// Mitsubishi GX Works2 project: PLS_programfiler_v1.0   PLC: FX2N/FX2NC

// global labels: Global1
VAR_GLOBAL
  Temperaturliste AT D0 : ARRAY [0..49] OF INT;
END_VAR

// task Task_01 (event TRUE, interval 0, priority 31): 

PROGRAM Kap7_765
(* structured ladder/FBD written out as ST: instructions are called as NAME(EN, inputs, outputs); _pN, _eN, _tN stand for wires *)
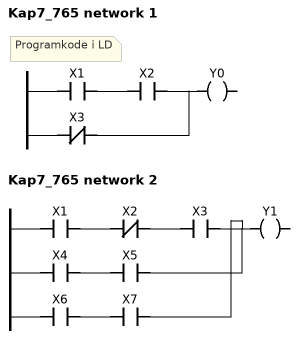
(* network 1 *)
(* Programkode i LD *)
Y0 := (X1 AND X2) OR (NOT X3);
(* network 2 *)
Y1 := (X1 AND NOT X2 AND X3) OR (X4 AND X5) OR (X6 AND X7);
END_PROGRAM

PROGRAM Kap7_766
(* structured ladder/FBD written out as ST: instructions are called as NAME(EN, inputs, outputs); _pN, _eN, _tN stand for wires *)
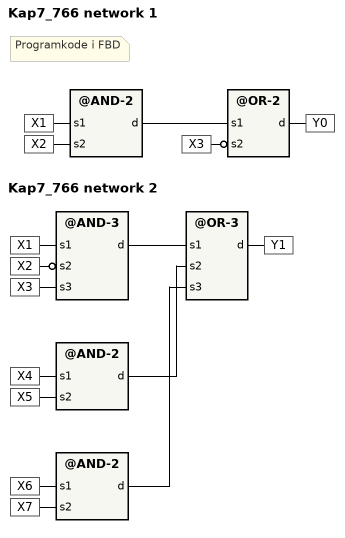
(* network 1 *)
(* Programkode i FBD *)
Y0 := @OR-2(@AND-2(X1, X2), NOT X3);
(* network 2 *)
Y1 := @OR-3(@AND-3(X1, NOT X2, X3), @AND-2(X4, X5), @AND-2(X6, X7));
END_PROGRAM

PROGRAM Kap7_768
(*Programkode i ST*)
Y0:=(X1 AND X2) OR NOT X3;
Y1:=(X1 AND NOT X2 AND X3) OR (X4 AND X5) OR (X6 AND X7);
END_PROGRAM

PROGRAM Kap7_764_IL
// body in language c0 not rendered
END_PROGRAM

PROGRAM Kap7_764_Melsec_IL
// body in language c0 not rendered
END_PROGRAM

FUNCTION Kap_7113_7114
VAR_INPUT
  Faktor1 : INT;
  Faktor2 : INT;
  Divisor : INT;
END_VAR
(* structured ladder/FBD written out as ST: instructions are called as NAME(EN, inputs, outputs); _pN, _eN, _tN stand for wires *)
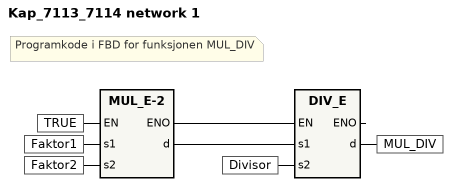
(* network 1 *)
(* Programkode i FBD for funksjonen MUL_DIV *)
_e2 := MUL_E(TRUE, Faktor1, Faktor2, _t1);
DIV_E(_e2, _t1, Divisor, MUL_DIV);
END_FUNCTION

FUNCTION_BLOCK Kap7_7103_7104
VAR_INPUT
  Start : BOOL;
  Stopp : BOOL;
  Motorvern : BOOL;
END_VAR
VAR_OUTPUT
  Motor : BOOL;
END_VAR
(* structured ladder/FBD written out as ST: instructions are called as NAME(EN, inputs, outputs); _pN, _eN, _tN stand for wires *)
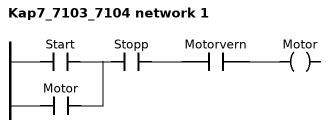
(* network 1 *)
Motor := ((Start OR Motor) AND Stopp) AND Motorvern;
END_FUNCTION_BLOCK

PROGRAM Kap4_481
(* structured ladder/FBD written out as ST: instructions are called as NAME(EN, inputs, outputs); _pN, _eN, _tN stand for wires *)
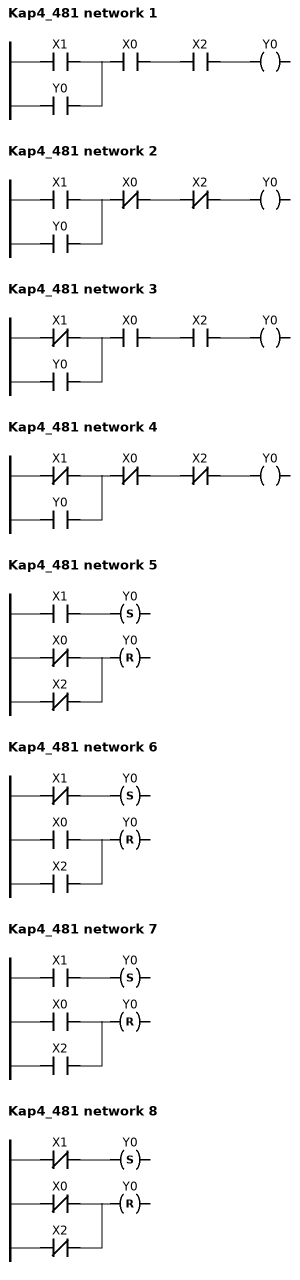
(* network 1 *)
Y0 := ((X1 OR Y0) AND X0) AND X2;
(* network 2 *)
Y0 := ((X1 OR Y0) AND NOT X0) AND NOT X2;
(* network 3 *)
Y0 := (((NOT X1) OR Y0) AND X0) AND X2;
(* network 4 *)
Y0 := (((NOT X1) OR Y0) AND NOT X0) AND NOT X2;
(* network 5 *)
SET(X1, Y0);
RST((NOT X0) OR (NOT X2), Y0);
(* network 6 *)
SET(NOT X1, Y0);
RST(X0 OR X2, Y0);
(* network 7 *)
SET(X1, Y0);
RST(X0 OR X2, Y0);
(* network 8 *)
SET(NOT X1, Y0);
RST((NOT X0) OR (NOT X2), Y0);
END_PROGRAM

PROGRAM Kap3_321
(* structured ladder/FBD written out as ST: instructions are called as NAME(EN, inputs, outputs); _pN, _eN, _tN stand for wires *)
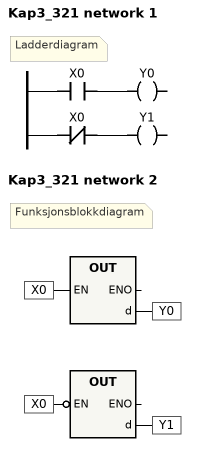
(* network 1 *)
(* Ladderdiagram *)
Y0 := X0;
Y1 := NOT X0;
(* network 2 *)
(* Funksjonsblokkdiagram *)
OUT(X0, Y0);
OUT(NOT X0, Y1);
END_PROGRAM

PROGRAM Kap3_322
(* structured ladder/FBD written out as ST: instructions are called as NAME(EN, inputs, outputs); _pN, _eN, _tN stand for wires *)
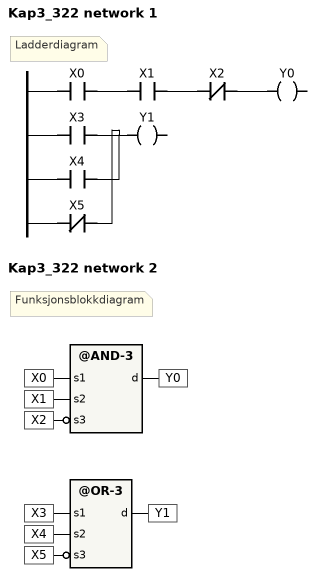
(* network 1 *)
(* Ladderdiagram *)
Y0 := X0 AND X1 AND NOT X2;
Y1 := X3 OR X4 OR (NOT X5);
(* network 2 *)
(* Funksjonsblokkdiagram *)
Y0 := @AND-3(X0, X1, NOT X2);
Y1 := @OR-3(X3, X4, NOT X5);
END_PROGRAM

PROGRAM Kap3_323
(* structured ladder/FBD written out as ST: instructions are called as NAME(EN, inputs, outputs); _pN, _eN, _tN stand for wires *)
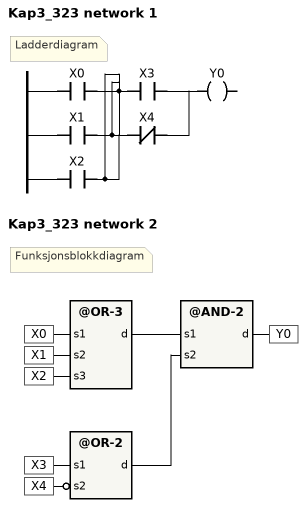
(* network 1 *)
(* Ladderdiagram *)
_p1 := X0 OR X1 OR X2;
Y0 := (_p1 AND X3) OR (_p1 AND NOT X4);
(* network 2 *)
(* Funksjonsblokkdiagram *)
Y0 := @AND-2(@OR-3(X0, X1, X2), @OR-2(X3, NOT X4));
END_PROGRAM

PROGRAM Kap3_324
(* structured ladder/FBD written out as ST: instructions are called as NAME(EN, inputs, outputs); _pN, _eN, _tN stand for wires *)
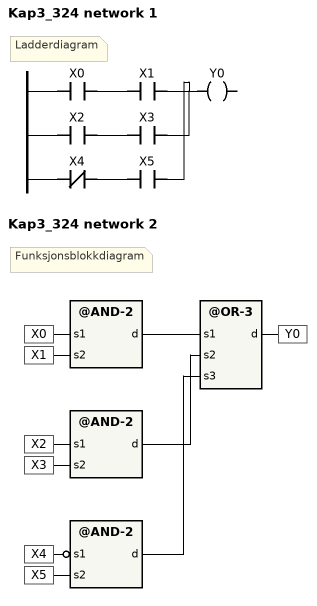
(* network 1 *)
(* Ladderdiagram *)
Y0 := (X0 AND X1) OR (X2 AND X3) OR (NOT X4 AND X5);
(* network 2 *)
(* Funksjonsblokkdiagram *)
Y0 := @OR-3(@AND-2(X0, X1), @AND-2(X2, X3), @AND-2(NOT X4, X5));
END_PROGRAM

PROGRAM Kap3_325
(* structured ladder/FBD written out as ST: instructions are called as NAME(EN, inputs, outputs); _pN, _eN, _tN stand for wires *)
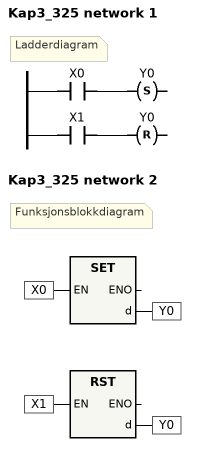
(* network 1 *)
(* Ladderdiagram *)
SET(X0, Y0);
RST(X1, Y0);
(* network 2 *)
(* Funksjonsblokkdiagram *)
SET(X0, Y0);
RST(X1, Y0);
END_PROGRAM

PROGRAM Kap3_326
(* structured ladder/FBD written out as ST: instructions are called as NAME(EN, inputs, outputs); _pN, _eN, _tN stand for wires *)
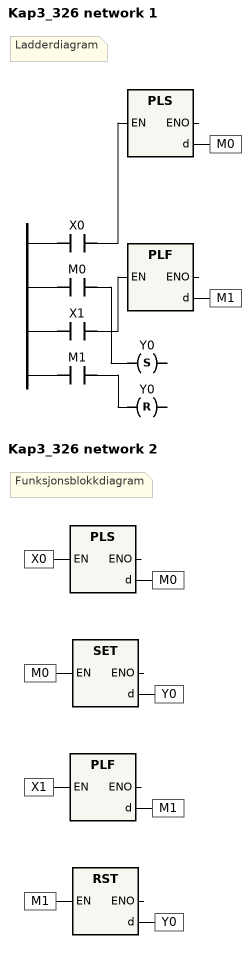
(* network 1 *)
(* Ladderdiagram *)
PLS(X0, M0);
SET(M0, Y0);
PLF(X1, M1);
RST(M1, Y0);
(* network 2 *)
(* Funksjonsblokkdiagram *)
PLS(X0, M0);
SET(M0, Y0);
PLF(X1, M1);
RST(M1, Y0);
END_PROGRAM

PROGRAM Kap3_336
(* structured ladder/FBD written out as ST: instructions are called as NAME(EN, inputs, outputs); _pN, _eN, _tN stand for wires *)
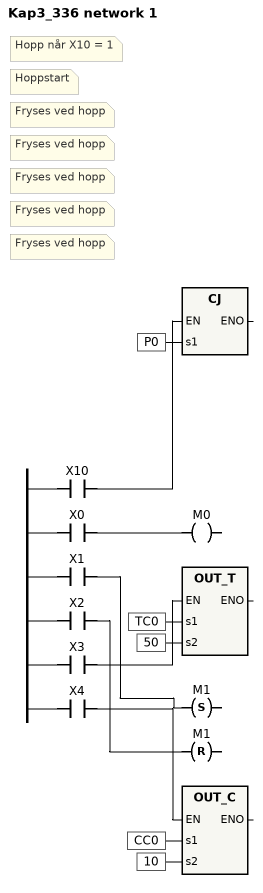
(* network 1 *)
(* Hopp når X10 = 1 *)
(* Hoppstart *)
(* Fryses ved hopp *)
(* Fryses ved hopp *)
(* Fryses ved hopp *)
(* Fryses ved hopp *)
(* Fryses ved hopp *)
CJ(X10, P0);
M0 := X0;
SET(X1, M1);
RST(X2, M1);
OUT_T(X3, TC0, 50);
OUT_C(X4, CC0, 10);
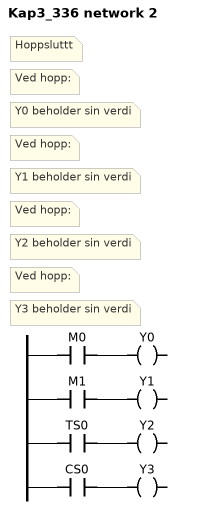
(* network 2 P0: *)
(* Hoppsluttt *)
(* Ved hopp: *)
(* Y0 beholder sin verdi *)
(* Ved hopp: *)
(* Y1 beholder sin verdi *)
(* Ved hopp: *)
(* Y2 beholder sin verdi *)
(* Ved hopp: *)
(* Y3 beholder sin verdi *)
Y0 := M0;
Y1 := M1;
Y2 := TS0;
Y3 := CS0;
END_PROGRAM

PROGRAM Kap5_5421
(* structured ladder/FBD written out as ST: instructions are called as NAME(EN, inputs, outputs); _pN, _eN, _tN stand for wires *)
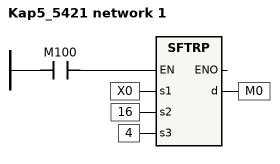
(* network 1 *)
SFTRP(M100, X0, 16, 4, M0);
END_PROGRAM

PROGRAM Kap3_331
(* structured ladder/FBD written out as ST: instructions are called as NAME(EN, inputs, outputs); _pN, _eN, _tN stand for wires *)
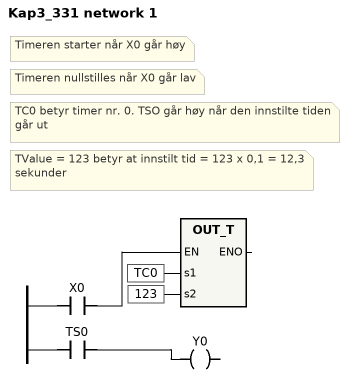
(* network 1 *)
(* Timeren starter når X0 går høy *)
(* Timeren nullstilles når X0 går lav *)
(* TC0 betyr timer nr. 0. TSO går høy når den innstilte tiden går ut *)
(* TValue = 123 betyr at innstilt tid = 123 x 0,1 = 12,3 sekunder *)
OUT_T(X0, TC0, 123);
Y0 := TS0;
END_PROGRAM

PROGRAM Kap3_333
(* structured ladder/FBD written out as ST: instructions are called as NAME(EN, inputs, outputs); _pN, _eN, _tN stand for wires *)
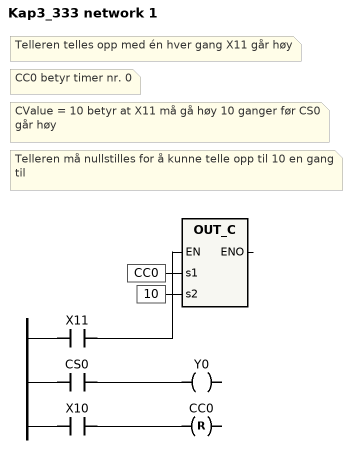
(* network 1 *)
(* Telleren telles opp med én hver gang X11 går høy *)
(* CC0 betyr timer nr. 0 *)
(* CValue = 10 betyr at X11 må gå høy 10 ganger før CS0 går høy *)
(* Telleren må nullstilles for å kunne telle opp til 10 en gang til *)
OUT_C(X11, CC0, 10);
Y0 := CS0;
RST(X10, CC0);
END_PROGRAM

PROGRAM Kap4_421
(* structured ladder/FBD written out as ST: instructions are called as NAME(EN, inputs, outputs); _pN, _eN, _tN stand for wires *)
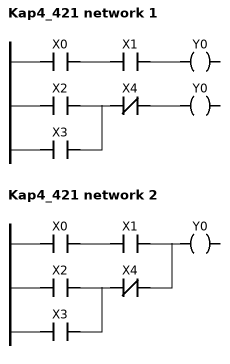
(* network 1 *)
Y0 := X0 AND X1;
Y0 := (X2 OR X3) AND NOT X4;
(* network 2 *)
Y0 := (X0 AND X1) OR ((X2 OR X3) AND NOT X4);
END_PROGRAM

PROGRAM Kap4_431
(* structured ladder/FBD written out as ST: instructions are called as NAME(EN, inputs, outputs); _pN, _eN, _tN stand for wires *)
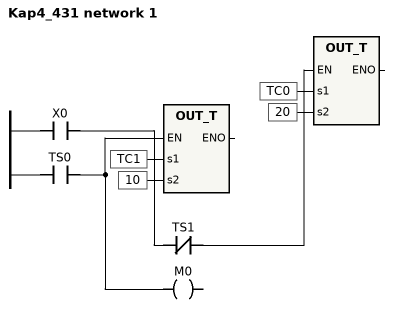
(* network 1 *)
OUT_T(X0 AND NOT TS1, TC0, 20);
OUT_T(TS0, TC1, 10);
M0 := TS0;
END_PROGRAM

PROGRAM Kap5_536_537
(* structured ladder/FBD written out as ST: instructions are called as NAME(EN, inputs, outputs); _pN, _eN, _tN stand for wires *)
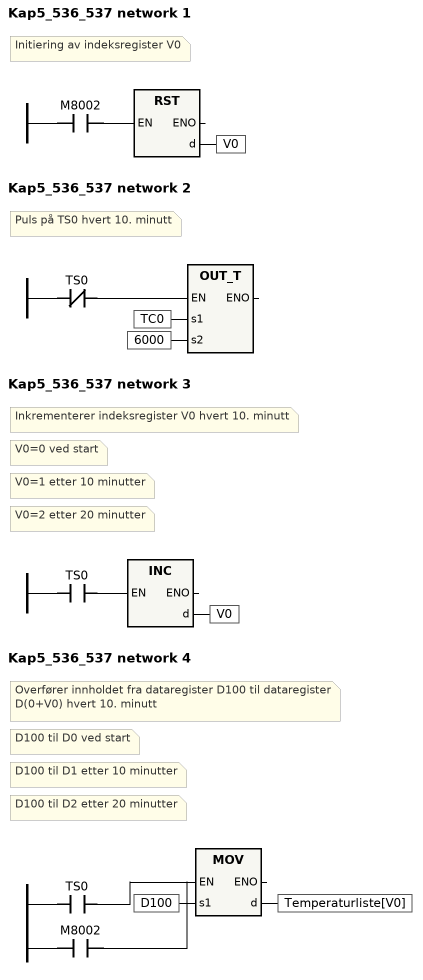
(* network 1 *)
(* Initiering av indeksregister V0 *)
RST(M8002, V0);
(* network 2 *)
(* Puls på TS0 hvert 10. minutt *)
OUT_T(NOT TS0, TC0, 6000);
(* network 3 *)
(* Inkrementerer indeksregister V0 hvert 10. minutt *)
(* V0=0 ved start *)
(* V0=1 etter 10 minutter *)
(* V0=2 etter 20 minutter *)
INC(TS0, V0);
(* network 4 *)
(* Overfører innholdet fra dataregister D100 til dataregister D(0+V0) hvert 10. minutt *)
(* D100 til D0 ved start *)
(* D100 til D1 etter 10 minutter *)
(* D100 til D2 etter 20 minutter *)
MOV(TS0 OR M8002, D100, Temperaturliste[V0]);
END_PROGRAM

PROGRAM Kap3_335
(* structured ladder/FBD written out as ST: instructions are called as NAME(EN, inputs, outputs); _pN, _eN, _tN stand for wires *)
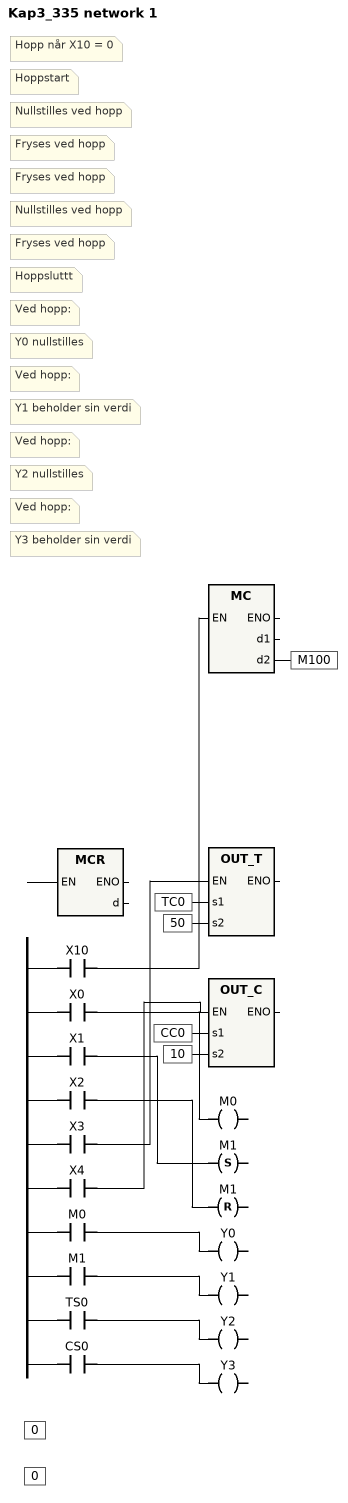
(* network 1 *)
(* Hopp når X10 = 0 *)
(* Hoppstart *)
(* Nullstilles ved hopp *)
(* Fryses ved hopp *)
(* Fryses ved hopp *)
(* Nullstilles ved hopp *)
(* Fryses ved hopp *)
(* Hoppsluttt *)
(* Ved hopp: *)
(* Y0 nullstilles *)
(* Ved hopp: *)
(* Y1 beholder sin verdi *)
(* Ved hopp: *)
(* Y2 nullstilles *)
(* Ved hopp: *)
(* Y3 beholder sin verdi *)
MC(X10, _open, M100);
M0 := X0;
SET(X1, M1);
RST(X2, M1);
OUT_T(X3, TC0, 50);
OUT_C(X4, CC0, 10);
MCR(TRUE, _open);
Y0 := M0;
Y1 := M1;
Y2 := TS0;
Y3 := CS0;
(* not connected to any output: 0, 0 *)
END_PROGRAM

PROGRAM Kap7_735
(* structured ladder/FBD written out as ST: instructions are called as NAME(EN, inputs, outputs); _pN, _eN, _tN stand for wires *)
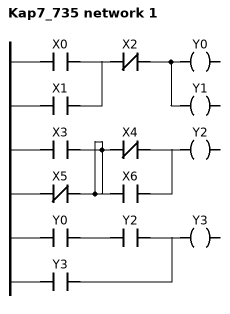
(* network 1 *)
_p1 := (X0 OR X1) AND NOT X2;
Y0 := _p1;
Y1 := _p1;
_p2 := X3 OR (NOT X5);
Y2 := (_p2 AND NOT X4) OR (_p2 AND X6);
Y3 := (Y0 AND Y2) OR Y3;
END_PROGRAM

PROGRAM Kap6_624
(* structured ladder/FBD written out as ST: instructions are called as NAME(EN, inputs, outputs); _pN, _eN, _tN stand for wires *)
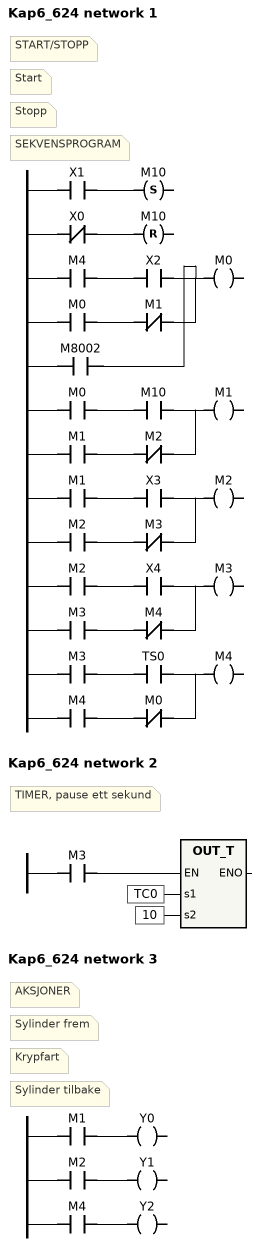
(* network 1 *)
(* START/STOPP *)
(* Start *)
(* Stopp *)
(* SEKVENSPROGRAM *)
SET(X1, M10);
RST(NOT X0, M10);
M0 := (M4 AND X2) OR (M0 AND NOT M1) OR M8002;
M1 := (M0 AND M10) OR (M1 AND NOT M2);
M2 := (M1 AND X3) OR (M2 AND NOT M3);
M3 := (M2 AND X4) OR (M3 AND NOT M4);
M4 := (M3 AND TS0) OR (M4 AND NOT M0);
(* network 2 *)
(* TIMER, pause ett sekund *)
OUT_T(M3, TC0, 10);
(* network 3 *)
(* AKSJONER *)
(* Sylinder frem *)
(* Krypfart *)
(* Sylinder tilbake *)
Y0 := M1;
Y1 := M2;
Y2 := M4;
END_PROGRAM

PROGRAM Kap6_625
(* structured ladder/FBD written out as ST: instructions are called as NAME(EN, inputs, outputs); _pN, _eN, _tN stand for wires *)
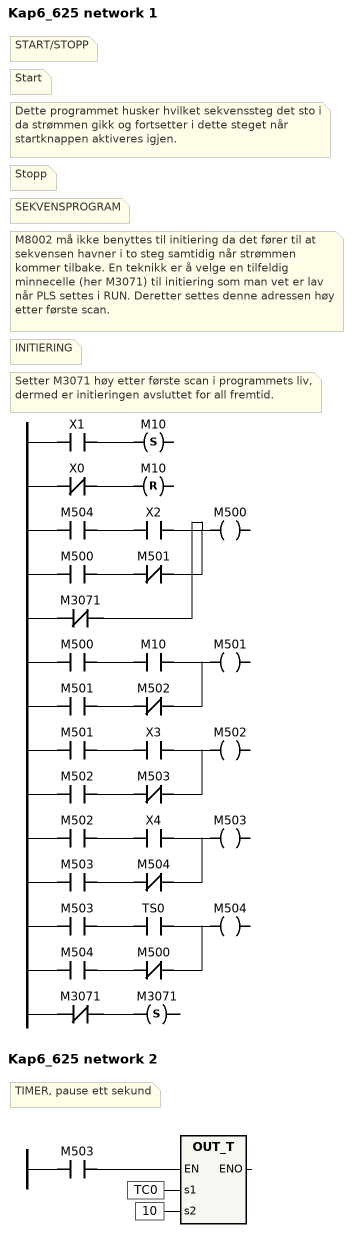
(* network 1 *)
(* START/STOPP *)
(* Start *)
(* Dette programmet husker hvilket sekvenssteg det sto i da strømmen gikk og fortsetter i dette steget når startknappen aktiveres igjen. *)
(* Stopp *)
(* SEKVENSPROGRAM *)
(* M8002 må ikke benyttes til initiering da det fører til at sekvensen havner i to steg samtidig når strømmen kommer tilbake. En teknikk er å velge en tilfeldig minnecelle (her M3071) til initiering som man vet er lav når PLS settes i RUN. Deretter settes denne adressen høy etter første scan. *)
(* INITIERING *)
(* Setter M3071 høy etter første scan i programmets liv, dermed er initieringen avsluttet for all fremtid. *)
SET(X1, M10);
RST(NOT X0, M10);
M500 := (M504 AND X2) OR (M500 AND NOT M501) OR (NOT M3071);
M501 := (M500 AND M10) OR (M501 AND NOT M502);
M502 := (M501 AND X3) OR (M502 AND NOT M503);
M503 := (M502 AND X4) OR (M503 AND NOT M504);
M504 := (M503 AND TS0) OR (M504 AND NOT M500);
SET(NOT M3071, M3071);
(* network 2 *)
(* TIMER, pause ett sekund *)
OUT_T(M503, TC0, 10);
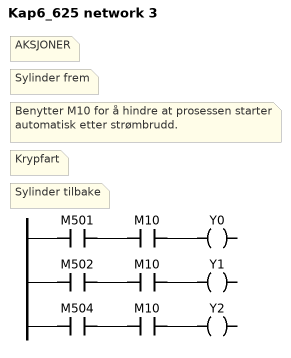
(* network 3 *)
(* AKSJONER *)
(* Sylinder frem *)
(* Benytter M10 for å hindre at prosessen starter automatisk etter strømbrudd. *)
(* Krypfart *)
(* Sylinder tilbake *)
Y0 := M501 AND M10;
Y1 := M502 AND M10;
Y2 := M504 AND M10;
END_PROGRAM

PROGRAM Kap6_632
(* structured ladder/FBD written out as ST: instructions are called as NAME(EN, inputs, outputs); _pN, _eN, _tN stand for wires *)
